{attribute 'qualified_only'}
{attribute 'strict'}
TYPE RecipeType_e :
(
    Smart := 0,
    Pro := 1,
    Mini := 2,
    Blue := 3,
    Smart_Kristall := 4,
    Pro_Smart := 5,
    Pro_Blue := 6,
    Pro_Smart_Kristall := 7,
    Pro_Smart_Maxi := 8,
    Pro_Smart_Maxi_Kristall := 9,
    Reserve := 10,
    _max
);
END_TYPE

(* stored: Version 1.1.0.1, ProductVersion 3.1.4024.6
   EnumerationTextList RecipeType_e: Id {4f8fe0cd-1876-4ea7-825f-c30cb68f3284} *)
